FUNCTION_BLOCK FB_Evacuador_SFC EXTENDS FB_Module_SFC
VAR_INPUT
    f0        : BOOL; (* gh0 (nombre=f0  c=I22 B=J2 b=22 módulo=EL1008 T=6  C=6 etiqueta=-B10, input) Pick and place de rechazo detrás *)
    f1        : BOOL; (* gh1 (nombre=f1  c=I23 B=J2 b=06 módulo=EL1008 T=6  C=6 etiqueta=-B11, input) Pick and place de rechazo delante *)
    g0        : BOOL; (* gv1 (nombre=g0  c=I24 B=J2 b=31 módulo=EL1008 T=6  C=6 etiqueta=-B12, input) Pick and place de rechazo arriba *)
    v1        : BOOL; (* ge1 (nombre=v1  c=I25 B=J1 b=25 módulo=EL1008 T=7  C=7 etiqueta=-B13, input) Pick and place de rechazo vacío *)
END_VAR
VAR_OUTPUT
    F_1       : BOOL; (* gHRA (nombre=F+  c=Q22 B=J2  b=35 módulo=EL2008 T=8 C=8 etiqueta=-Y8,  output) Pick and place de rechazo avanza (afuera) *)
    F_0       : BOOL; (* gHRR (nombre=F-  c=Q23 B=J2  b=32 módulo=EL2008 T=8 C=8 etiqueta=-Y9,  output) Pick and place de rechazo retrocede *)
    G_1       : BOOL; (* gVER (nombre=G+  c=Q24 B=J2  b=11 módulo=EL2008 T=8 C=8 etiqueta=-Y10, output) Pick and place de rechazo baja *)
    V_1       : BOOL; (* gEYE (nombre=V+  c=Q25 B=J2  b=08 módulo=EL2008 T=9 C=9 etiqueta=-Y11, output) Pick and place de rechazo succiona *)
END_VAR
VAR
END_VAR

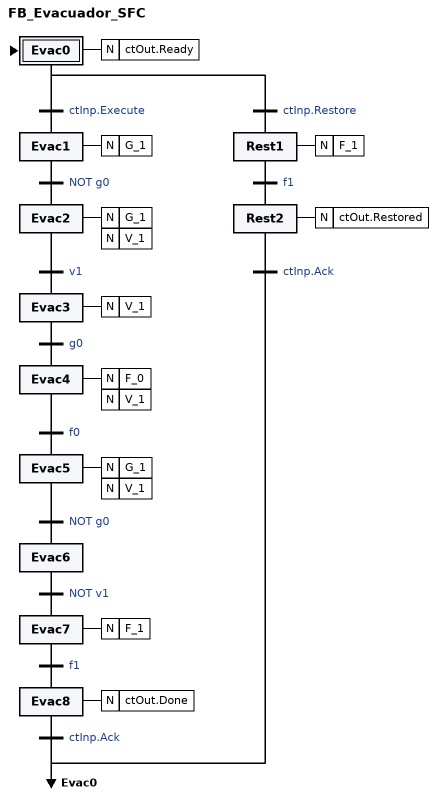
INITIAL_STEP Evac0:
    ctOut.Ready(N);
END_STEP
TRANSITION FROM Evac0 TO Evac1
    := ctInp.Execute;
END_TRANSITION
STEP Evac1:
    G_1(N);
END_STEP
TRANSITION FROM Evac1 TO Evac2
    := NOT g0;
END_TRANSITION
STEP Evac2:
    G_1(N);
    V_1(N);
END_STEP
TRANSITION FROM Evac2 TO Evac3
    := v1;
END_TRANSITION
STEP Evac3:
    V_1(N);
END_STEP
TRANSITION FROM Evac3 TO Evac4
    := g0;
END_TRANSITION
STEP Evac4:
    F_0(N);
    V_1(N);
END_STEP
TRANSITION FROM Evac4 TO Evac5
    := f0;
END_TRANSITION
STEP Evac5:
    G_1(N);
    V_1(N);
END_STEP
TRANSITION FROM Evac5 TO Evac6
    := NOT g0;
END_TRANSITION
STEP Evac6:
END_STEP
TRANSITION FROM Evac6 TO Evac7
    := NOT v1;
END_TRANSITION
STEP Evac7:
    F_1(N);
END_STEP
TRANSITION FROM Evac7 TO Evac8
    := f1;
END_TRANSITION
STEP Evac8:
    ctOut.Done(N);
END_STEP
TRANSITION FROM Evac8 TO Evac0
    := ctInp.Ack;
END_TRANSITION
TRANSITION FROM Evac0 TO Rest1
    := ctInp.Restore;
END_TRANSITION
STEP Rest1:
    F_1(N);
END_STEP
TRANSITION FROM Rest1 TO Rest2
    := f1;
END_TRANSITION
STEP Rest2:
    ctOut.Restored(N);
END_STEP
TRANSITION FROM Rest2 TO Evac0
    := ctInp.Ack;
END_TRANSITION

END_FUNCTION_BLOCK

(* stored: Version 1.1.0.1, ProductVersion 3.1.4024.11
   POU FB_Evacuador_SFC: Id {732a5d89-d610-4122-b553-0a1448cdc8d0}, SpecialFunc None *)
